// Mitsubishi GX Works2 project: servo_block_loop   PLC: Q02/Q02H

PROGRAM MAIN
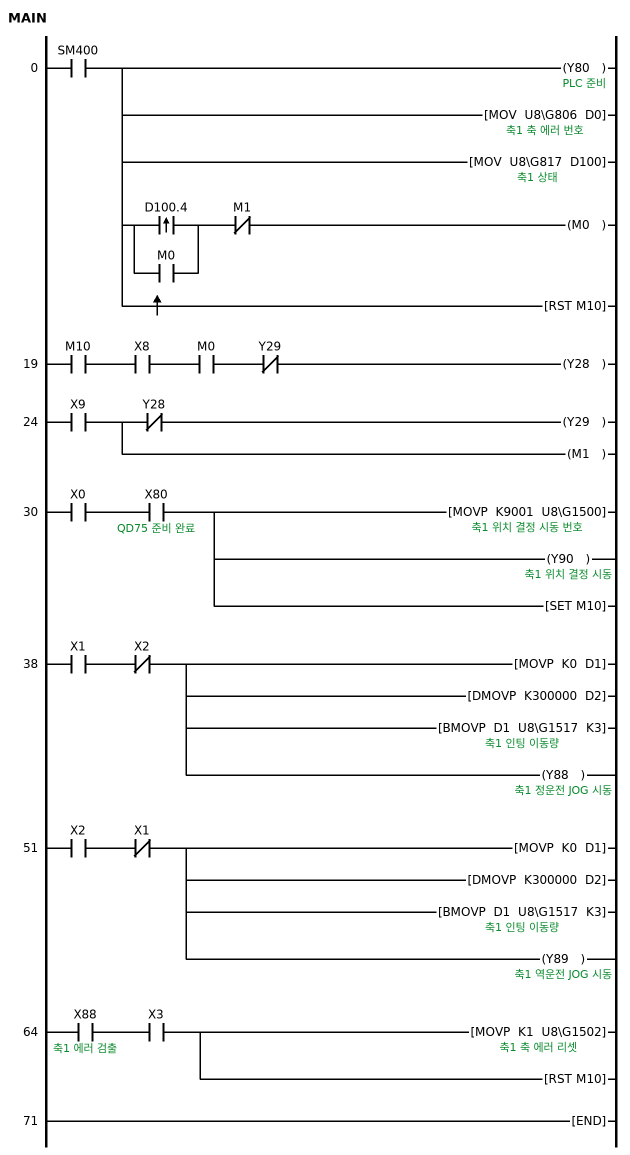
0     LD      SM400
      OUT     Y80  ; PLC 준비
      MOV     U8\G806 D0  ; 축1 축 에러 번호
      MOV     U8\G817 D100  ; 축1 상태
      MPS
      LDP     D100.4
      OR      M0
      ANB
      ANI     M1
      OUT     M0
      MPP
      MEP
      RST     M10
19    LD      M10
      AND     X8
      AND     M0
      ANI     Y29
      OUT     Y28
24    LD      X9
      MPS
      ANI     Y28
      OUT     Y29
      MPP
      OUT     M1
30    LD      X0
      AND     X80  ; QD75 준비 완료
      MOVP    K9001 U8\G1500  ; 축1 위치 결정 시동 번호
      OUT     Y90  ; 축1 위치 결정 시동
      SET     M10
38    LD      X1
      ANI     X2
      MOVP    K0 D1
      DMOVP   K300000 D2
      BMOVP   D1 U8\G1517 K3  ; 축1 인팅 이동량
      OUT     Y88  ; 축1 정운전 JOG 시동
51    LD      X2
      ANI     X1
      MOVP    K0 D1
      DMOVP   K300000 D2
      BMOVP   D1 U8\G1517 K3
      OUT     Y89  ; 축1 역운전 JOG 시동
64    LD      X88  ; 축1 에러 검출
      AND     X3
      MOVP    K1 U8\G1502  ; 축1 축 에러 리셋
      RST     M10
71    END
END_PROGRAM

PROGRAM MAIN1
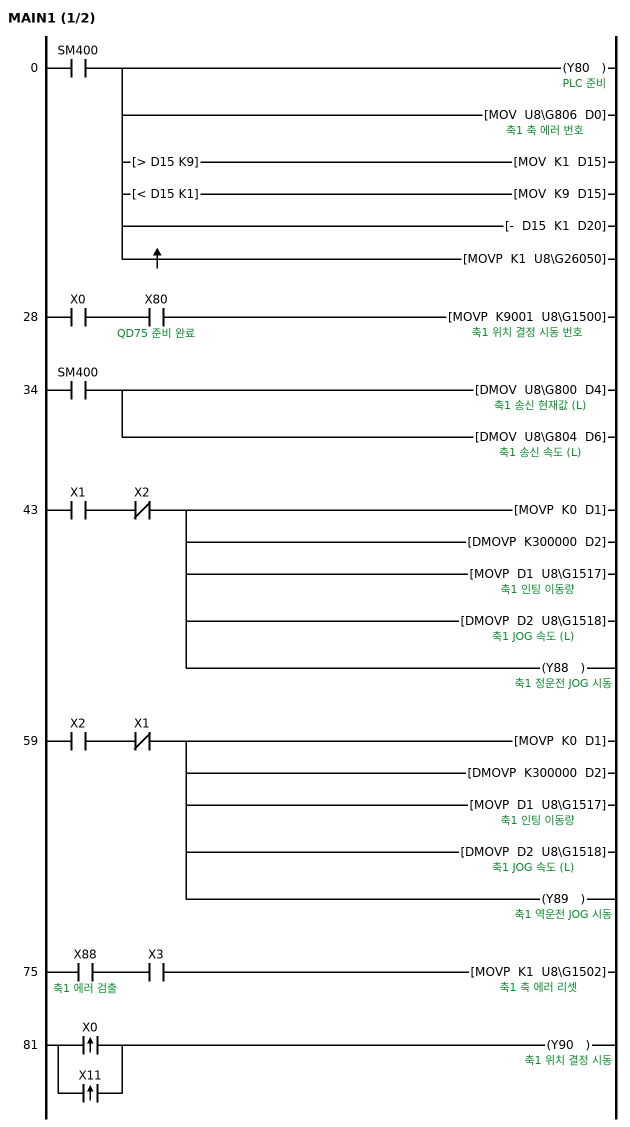
0     LD      SM400
      OUT     Y80  ; PLC 준비
      MOV     U8\G806 D0  ; 축1 축 에러 번호
      MPS
      AND>    D15 K9
      MOV     K1 D15
      MRD
      AND<    D15 K1
      MOV     K9 D15
      MPP
      -       D15 K1 D20
      MEP
      MOVP    K1 U8\G26050
28    LD      X0
      AND     X80  ; QD75 준비 완료
      MOVP    K9001 U8\G1500  ; 축1 위치 결정 시동 번호
34    LD      SM400
      DMOV    U8\G800 D4  ; 축1 송신 현재값 (L)
      DMOV    U8\G804 D6  ; 축1 송신 속도 (L)
43    LD      X1
      ANI     X2
      MOVP    K0 D1
      DMOVP   K300000 D2
      MOVP    D1 U8\G1517  ; 축1 인팅 이동량
      DMOVP   D2 U8\G1518  ; 축1 JOG 속도 (L)
      OUT     Y88  ; 축1 정운전 JOG 시동
59    LD      X2
      ANI     X1
      MOVP    K0 D1
      DMOVP   K300000 D2
      MOVP    D1 U8\G1517
      DMOVP   D2 U8\G1518
      OUT     Y89  ; 축1 역운전 JOG 시동
75    LD      X88  ; 축1 에러 검출
      AND     X3
      MOVP    K1 U8\G1502  ; 축1 축 에러 리셋
81    LDP     X0
      ORP     X11
      OUT     Y90  ; 축1 위치 결정 시동
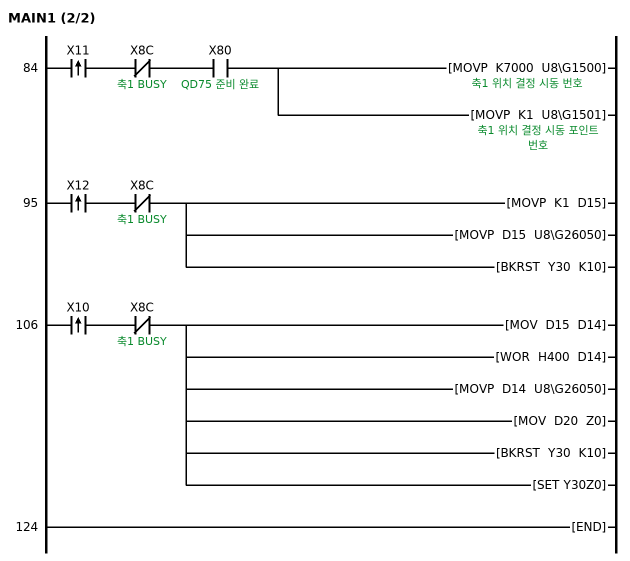
84    LDP     X11
      ANI     X8C  ; 축1 BUSY
      AND     X80  ; QD75 준비 완료
      MOVP    K7000 U8\G1500
      MOVP    K1 U8\G1501  ; 축1 위치 결정 시동 포인트 번호
95    LDP     X12
      ANI     X8C  ; 축1 BUSY
      MOVP    K1 D15
      MOVP    D15 U8\G26050
      BKRST   Y30 K10
106   LDP     X10
      ANI     X8C  ; 축1 BUSY
      MOV     D15 D14
      WOR     H400 D14
      MOVP    D14 U8\G26050
      MOV     D20 Z0
      BKRST   Y30 K10
      SET     Y30Z0
124   END
END_PROGRAM

// device comments not shown above
X81  ; 동기용 플래그
X84  ; 축1 M 코드 ON
X85  ; 축2 M 코드 ON
X89  ; 축2 에러 검출
X8D  ; 축2 BUSY
X90  ; 축1 시동 완료
X91  ; 축2 시동 완료
X94  ; 축1 위치 결정 완료
X95  ; 축2 위치 결정 완료
Y84  ; 축1 축 정지
Y85  ; 축2 축 정지
Y8A  ; 축2 정운전 JOG 시동
Y8B  ; 축2 역운전 JOG 시동
Y91  ; 축2 위치 결정 시동
Y94  ; 축1 실행 금지 플래그
Y95  ; 축2 실행 금지 플래그
